_CFC_ (* Continuous Function Chart, elements in execution order *)
#0 AND(#6.out 7, SHU6_PV1_YARQ1_DI5_A)
#1 OR(SHU6_PV1_UST_RE_PUSK, SHU6_PV1_UST_RE_RABOTA)
#2 OR(SHU6_PV1_UST_RE_OSTANOV, SHU6_PV1_UST_RE_STOP)
#3 SR_VKL:SR(SET1: #1, RESET: #2)
#4 OR(SHU6_PV1_RQ1_DI3_ALM, SHU6_PV1_Z_MRQ1_NPIT)
#5 AND(SHU6_PV1_RQ1_DI3_RUN, SHU6_PV1_YARQ1_DI5_A)
#6 fb_HVACMS_M3:FB_HVACMotor1Speed(eHVACDataSecurityType_Idle, FALSE, TRUE, #3.Q1, eHVACActuatorMode_Auto_BMS, NOT #4, #5, NOT SHU6_PV1_Z_NETP_MRQ1, TRUE, TRUE, TRUE, SHU6_PV1_SB, startDelay_M3, stopDelay_M3, delayFBC_M3, feedbPT_M3, delayFBP_M3)
#7 SHU6_PV1_RQ1_DO5_VKL <= #6.out 1
#8 MRQ1_OTKAZ <= #0
#9 INT_TO_TIME(SHU6_PV1_M_TI)
#10 MUL(#9, 1000)
#11 tTi <= #10
_END_CFC_
END_PROGRAM

(* POU IM/RQ1_CHASTOTA, CFC *)
PROGRAM RQ1_CHASTOTA
VAR
	RQ1_PID: FB_HVACPIDCtrl;

          deadRange: REAL := 0.1;
	direction: BOOL;



         tTi: TIME;
	tTv: TIME;
	tTd: TIME:=T#0s;
         rYMin: REAL := 30;
         rYMax: REAL := 48;
	CHASTOTA_RQ1: RAMP_REAL;
	FT_MANUAL_RQ1: F_TRIG;
	RT_AVT_RQ1: R_TRIG;
	RS_REG_UPR_RQ1: RS;
END_VAR
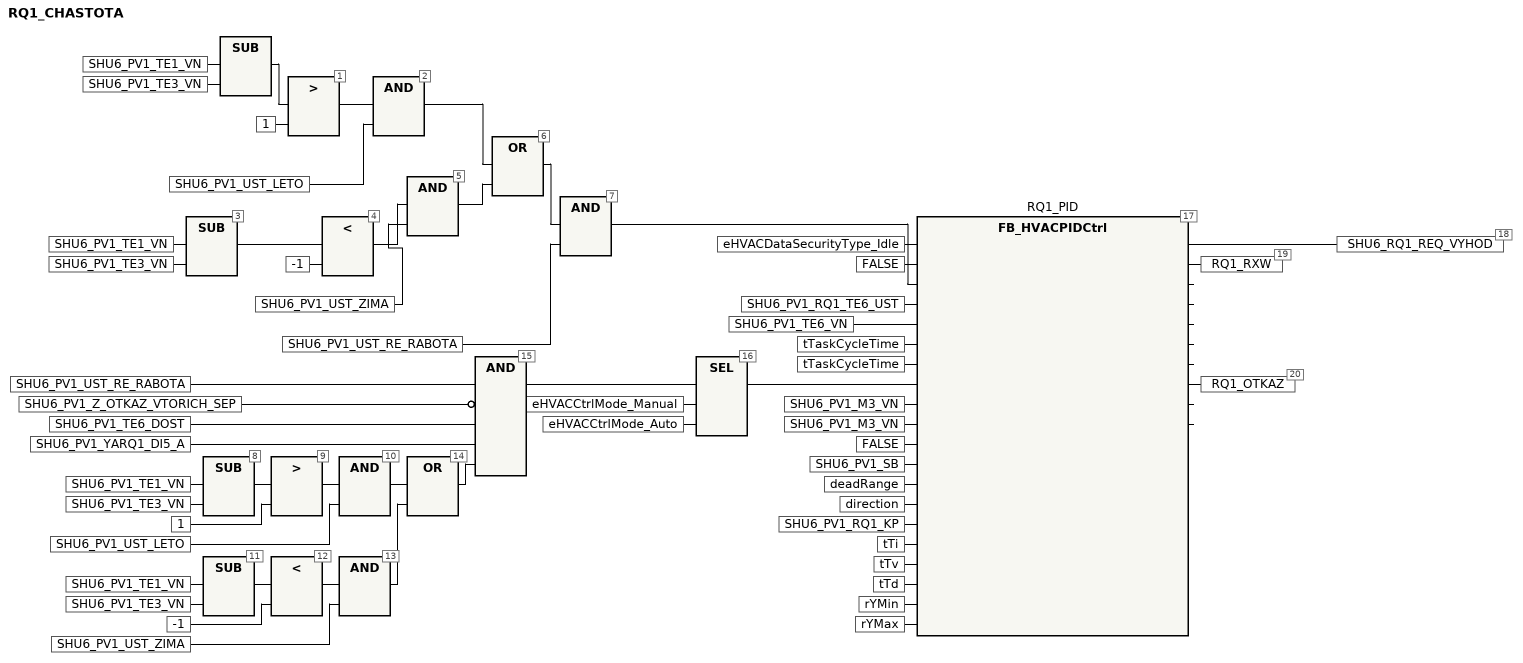
_CFC_ (* Continuous Function Chart, elements in execution order *)
#0 SUB(SHU6_PV1_TE1_VN, SHU6_PV1_TE3_VN)
#1 >(#0, 1)
#2 AND(#1, SHU6_PV1_UST_LETO)
#3 SUB(SHU6_PV1_TE1_VN, SHU6_PV1_TE3_VN)
#4 <(#3, -1)
#5 AND(#4, SHU6_PV1_UST_ZIMA)
#6 OR(#2, #5)
#7 AND(#6, SHU6_PV1_UST_RE_RABOTA)
#8 SUB(SHU6_PV1_TE1_VN, SHU6_PV1_TE3_VN)
#9 >(#8, 1)
#10 AND(#9, SHU6_PV1_UST_LETO)
#11 SUB(SHU6_PV1_TE1_VN, SHU6_PV1_TE3_VN)
#12 <(#11, -1)
#13 AND(#12, SHU6_PV1_UST_ZIMA)
#14 OR(#10, #13)
#15 AND(SHU6_PV1_UST_RE_RABOTA, NOT SHU6_PV1_Z_OTKAZ_VTORICH_SEP, SHU6_PV1_TE6_DOST, SHU6_PV1_YARQ1_DI5_A, #14)
#16 SEL(#15, eHVACCtrlMode_Manual, eHVACCtrlMode_Auto)
#17 RQ1_PID:FB_HVACPIDCtrl(eHVACDataSecurityType_Idle, FALSE, #7, SHU6_PV1_RQ1_TE6_UST, SHU6_PV1_TE6_VN, tTaskCycleTime, tTaskCycleTime, #16, SHU6_PV1_M3_VN, SHU6_PV1_M3_VN, FALSE, SHU6_PV1_SB, deadRange, direction, SHU6_PV1_RQ1_KP, tTi, tTv, tTd, rYMin, rYMax)
#18 SHU6_RQ1_REQ_VYHOD <= #17.out 1
#19 RQ1_RXW <= #17.out 2
#20 RQ1_OTKAZ <= #17.out 8
_END_CFC_
END_PROGRAM

(* POU IM/YA1_Upr, CFC *)
PROGRAM YA1_Upr
VAR
        enableLimitSwitch: BOOL := TRUE;
        stokeTime: TIME;
	RS_YA1_OPEN: RS;
	RT_PUSK: R_TRIG;
       TON_PCH_OTKL: TON;
	RT_PCH_OTKL: R_TRIG;
	fb_HVACPAYa1: FB_HVAC2PointActuator;
END_VAR
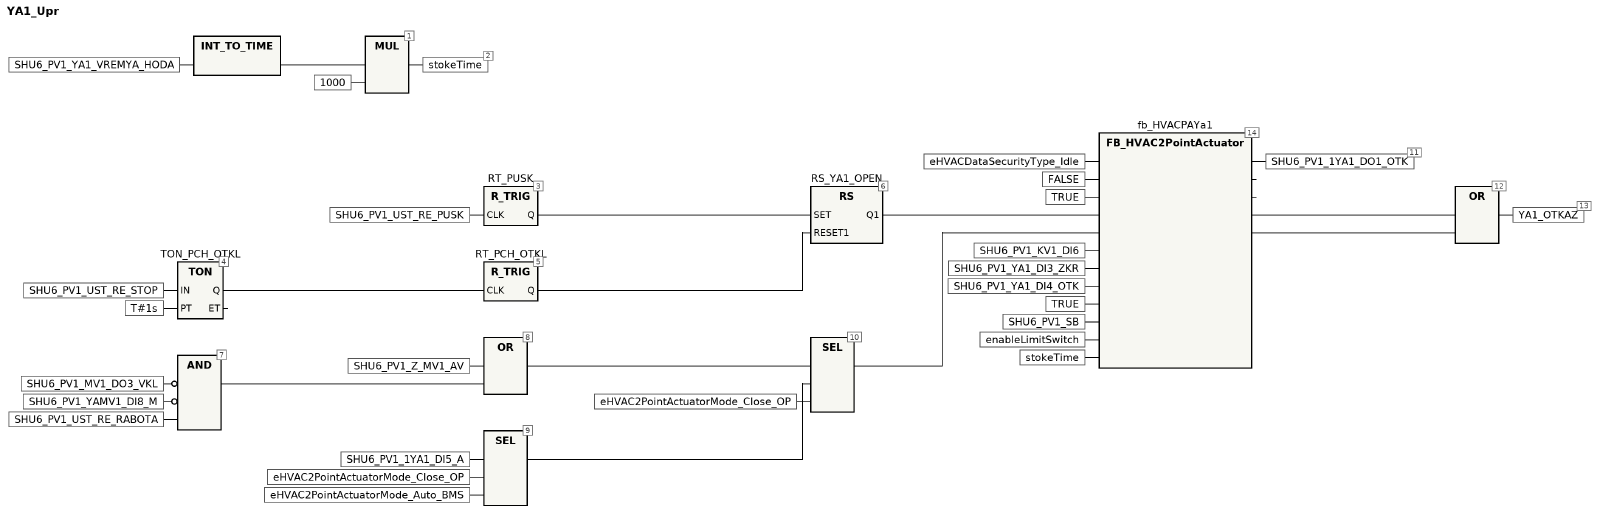
